// TwinCAT 3 PLC project Untitled3
// ProgramVersion: 3.1.4026.18
// libraries:
//   Tc2_EtherCAT, * (Beckhoff Automation GmbH)
//   Tc2_MC2, * (Beckhoff Automation GmbH)
//   Tc2_Standard, * (Beckhoff Automation GmbH)
//   Tc2_System, * (Beckhoff Automation GmbH)
//   Tc3_EtherCATDiag, * (Beckhoff Automation GmbH)
//   Tc3_EventLogger, * (Beckhoff Automation GmbH)
//   Tc3_Module, * (Beckhoff Automation GmbH)
// project tree:
//   DUTs/ E_SignalMode.TcDUT, ST_TsDiagObjectsEL1904.TcDUT, ST_TsDiagObjectsEL2904.TcDUT, ST_TsDiagObjectsEL1918.TcDUT, ST_TsDiagObjectsEL2912.TcDUT
//   POUs/TwinSAFE FBs/ FB_CoEDiagObjects_EL1904.TcPOU, FB_CoEDiagObjects_EL1918.TcPOU (not stored), FB_CoEDiagObjects_EL2904.TcPOU (not stored), FB_CoEDiagObjects_EL2912.TcPOU (not stored), FB_TsConnection_Diag.TcPOU (not stored), FB_TsConnection_Diag_EL2912.TcPOU, FB_TsConnection_EtherCATState_EL2904.TcPOU, FB_TsConnection_EtherCATState_EL2912.TcPOU, FB_TsConnection_State.TcPOU (not stored), FB_TsConnection_EtherCatState_EL1918.TcPOU, FB_TsConnection_Diag_EL1918.TcPOU, FB_TsConnection_EtherCATState_EL1904.TcPOU (not stored), FB_TsFBEDM_Diag.TcPOU, FB_TsFBEDM_State.TcPOU, FB_TsFBEStop_Diag.TcPOU, FB_TsFBEStop_State.TcPOU (not stored), FB_TsFBMon_Diag.TcPOU (not stored), FB_TsFBMon_State.TcPOU, FB_TsGroup_Diag.TcPOU (not stored), FB_TsGroup_State.TcPOU (not stored)
//   POUs/ MAIN.TcPOU
//   / Test1.TcTTO
// real-time tasks:
//   TASK Test1: cycle T#10ms, priority 2, ADS port 350
// motion (NC):
//   TASK NC-Task 1 SAF NEW: cycle T#2ms, priority 4, ADS port 501
//   TASK NC-Task 1 SVB: cycle T#10ms, priority 8, ADS port 511
//   AXIS Axis 1 (id 1)
//     General: UnitName=°
//     Dynamic: Acceleration=15000, Deceleration=15000, Jerk=52947
//     Velo: RefSearch=117.66, RefSync=117.66, SlowManual=588.3, FastManual=3529.8, Fast=11766, Maximum=11766
//     OtherSettings: AllowMotionCmdToSlave=true
//     encoder EncType=19
//       EncPara: ScaleFactorNumerator=360, ScaleFactorDenominator=1048576, MaxCount=#xffffffff
//     drive DrvType=16
//       DrvPara: MaxCount=#xffffffff, DriveControlDWord=#x00020100
//         Analog: VeloReferenz=12942.6, VeloScale=32, TorqueSetpointScale=10, ScaleFactorActTorque=0.1
//         TimeComp: TaskDelayCycles=1
//     controller CtrType=1
//       CtrPara: PriorControlFactor=1
//         PosDiffControl: Range=50
//         Observer: BandWidth=20
//   AXIS Axis 2 (id 2)
//     General: UnitName=°
//     Dynamic: Acceleration=4263.1575, Deceleration=4263.1575, Jerk=12789.4725
//     Velo: RefSearch=28.42105, RefSync=28.42105, SlowManual=142.10525, FastManual=852.6315, Fast=2842.105, Maximum=2842.105
//     OtherSettings: AllowMotionCmdToSlave=true
//     encoder EncType=4
//       EncPara: ScaleFactorNumerator=360, ScaleFactorDenominator=4096, MaxCount=#x0000ffff
//         Inc: RefSoftSyncMask=#x0000ffff
//     drive DrvType=24
//       Analog: VeloReferenz=3600, TorqueSetpointScale=10, ScaleFactorActTorque=0.1
//       TimeComp: TaskDelayCycles=1
//     controller CtrType=1
//       CtrPara: PriorControlFactor=1
//         PosDiffControl: Range=50
//         Observer: BandWidth=20
// I/O:
//   DEVICE Device 1 (EtherCAT), AmsNetId 169.254.191.109.2.1
//     Term 19 (EK1200) [EK1200-5000 EtherCAT Power supply (2A E-Bus)]
//       Term 20 (EL1918) [EL1918, 8Ch. Safety Input 24V, TwinSAFE]
//         modules: Module 2 (FSLOGIC)
//       Term 21 (EL1904) [EL1904, 4 Ch. Safety Input 24V, TwinSAFE]
//         modules: Module 1 (FSOES)
//       Term 22 (EL2904) [EL2904, 4 Ch. Safety Output 24V, 0.5A, TwinSAFE]
//         modules: Module 1 (FSOES), Module 2 (DO)
//       Term 23 (EK1122) [EK1122 2 port EtherCAT junction]
//         Term 24 (EK1101) [EK1101 EtherCAT Coupler (2A E-Bus, ID switch)]
//           Term 25 (EL2912) [EL2912, 2Ch. Safety Output 24V, 2A, TwinSAFE]
//             modules: Module 1 (FSOE), Module 2 (FSOUT), Module 3 (DEVICEIO), Module 4 (FSLOGIC)
//           Term 26 (EK1122) [EK1122 2 port EtherCAT junction]
//             Term 27 (EK1101-0010) [EK1101-0010 EtherCAT Coupler (2A E-Bus, ID switch, Extended Distance)]
//               Term 28 (EL3074) [EL3074 4Ch. Ana. Input +/-10V, +/-20mA]
//               Term 29 (EL3174) [EL3174 4Ch. Ana. Input +/-10V Diff., +/-20mA SingleEnded, 16 Bit]
//               Term 30 (EL3202-0010) [EL3202-0010 2Ch. Ana. Input PT100 (RTD), High Precision]
//               Term 31 (ELM3142-0000) [ELM3142-0000 2Ch. Ana. Input +/-10V, +/-20mA, 24 bit, high precision]
//               Term 32 (EL4712) [EL4712 2Ch. Ana. Output 0-20mA, Oversample]
//               Term 33 (EL4732) [EL4732 2Ch. Ana. Output +/-10V, Oversample]
//               Term 34 (EL9510) [EL9510 Power supply terminal 10V]
//               Term 35 (EK1122) [EK1122 2 port EtherCAT junction]
//                 Term 36 (EK1100) [EK1100 EtherCAT Coupler (2A E-Bus)]
//                   Term 37 (EL7201-9014) [EL7201-9014 1Ch. MDP742 Servo motor output stage with OCT (50V, 2.8A RMS) and STO input]
//                     startup 32785:21 := 0E01 // DRV Motor Settings / Commutation offset
//                     startup 32785:27 := A9070000 // DRV Motor Settings / Motor speed limitation
//                     startup 28688:3 := 09 // DRV Outputs / Modes of operation
//                     startup 32784:87 := 64 // DRV Amplifier Settings / Velocity feed forward gain
//                     startup 28688:11 := 880B // DRV Outputs / Torque limitation
//                     startup 32784:19 := B200 // DRV Amplifier Settings / Current loop proportional gain
//                     startup 32784:18 := 0500 // DRV Amplifier Settings / Current loop integral time
//                     startup 32784:21 := 2B000000 // DRV Amplifier Settings / Velocity loop proportional gain
//                     startup 32784:20 := 96000000 // DRV Amplifier Settings / Velocity loop integral time
//                     startup 32768:1 := 00 // FB Settings / Invert feedback direction
//                   Term 38 (EL7037) [EL7037 1Ch. Stepper motor output stage (24V, 1.5A)]
//                     startup 32786:5 := 02 // STM Features Ch.1 / Speed range
//                     startup 32785:1 := DE01 // STM Controller Settings Ch.1 / Kp factor (curr.)
//                     startup 32785:2 := A200 // STM Controller Settings Ch.1 / Ki factor (curr.)
//                     startup 32788:3 := C0010000 // STM Controller Settings 3 Ch.1 / Kp factor (velo.)
//                     startup 32788:4 := 8813 // STM Controller Settings 3 Ch.1 / Tn (velo.)
//                     startup 32786:8 := 00 // STM Features Ch.1 / Feedback type
//                   Term 39 (EL9011) [EL9011 End Terminal]
// variable links:
//   Device 1 (EtherCAT) <-> Device 1 (EtherCAT)/Term 19 (EK1200)/Term 21 (EL1904)
//     Term 19 (EK1200)/Term 20 (EL1918)/ConnectionInputs/TwinSafeGroup1.Term 3 (EL1904) - Module 1 (FSOES)_4 TxPDO <-> Module 1 (FSOES)/RxPDO/FSOE
//     Term 19 (EK1200)/Term 20 (EL1918)/ConnectionOutputs/TwinSafeGroup1.Term 3 (EL1904) - Module 1 (FSOES)_4 RxPDO <-> Module 1 (FSOES)/TxPDO/FSOE
//   Device 1 (EtherCAT) <-> Device 1 (EtherCAT)/Term 19 (EK1200)/Term 22 (EL2904)
//     Term 19 (EK1200)/Term 20 (EL1918)/ConnectionInputs/TwinSafeGroup1.Term 4 (EL2904) - Module 1 (FSOES)_5 TxPDO <-> Module 1 (FSOES)/RxPDO/FSOE
//     Term 19 (EK1200)/Term 20 (EL1918)/ConnectionOutputs/TwinSafeGroup1.Term 4 (EL2904) - Module 1 (FSOES)_5 RxPDO <-> Module 1 (FSOES)/TxPDO/FSOE
//   Device 1 (EtherCAT) <-> Device 1 (EtherCAT)/Term 19 (EK1200)/Term 23 (EK1122)/Term 24 (EK1101)/Term 25 (EL2912)
//     Term 19 (EK1200)/Term 20 (EL1918)/ConnectionInputs/TwinSafeGroup1.Term 5 (EL2912) - Module 1 (FSOE)_6 TxPDO <-> Module 1 (FSOE)/FSoE Outputs/FSOE
//     Term 19 (EK1200)/Term 20 (EL1918)/ConnectionOutputs/TwinSafeGroup1.Term 5 (EL2912) - Module 1 (FSOE)_6 RxPDO <-> Module 1 (FSOE)/FSoE Inputs/FSOE
//   NC-Task 1 SAF NEW/Axes/Axis 1 <-> Device 1 (EtherCAT)/Term 19 (EK1200)/Term 23 (EK1122)/Term 24 (EK1101)/Term 26 (EK1122)/Term 27 (EK1101-0010)/Term 35 (EK1122)/Term 36 (EK1100)/Term 37 (EL7201-9014)
//     Drive/Inputs/In/nDataIn1 <-> DRV Following error actual value/Following error actual value
//     Drive/Inputs/In/nDataIn3[0] <-> DRV Torque actual value/Torque actual value
//     Drive/Inputs/In/nDcOutputTime <-> InfoData/DcOutputShift
//     Drive/Inputs/In/nState1 <-> DRV Statusword/Statusword
//     Drive/Inputs/In/nState2 <-> DRV Statusword/Statusword @bit 8
//     Drive/Inputs/In/nState4 @bit 1 <-> WcState/InputToggle
//     Drive/Inputs/In/nState4 <-> WcState/WcState
//     Drive/Outputs/Out/nCtrl1 <-> DRV Controlword/Controlword
//     Drive/Outputs/Out/nCtrl2 <-> DRV Controlword/Controlword @bit 8
//     Drive/Outputs/Out/nDataOut1 <-> DRV Target position/Target position
//     Drive/Outputs/Out/nDataOut2 <-> DRV Target velocity/Target velocity
//     Enc/Inputs/In/nDataIn1 <-> FB Position/Position
//     Enc/Inputs/In/nDcInputTime <-> InfoData/DcInputShift
//     Enc/Inputs/In/nState4 @bit 1 <-> WcState/InputToggle
//     Enc/Inputs/In/nState4 <-> WcState/WcState
//   NC-Task 1 SAF NEW/Axes/Axis 2 <-> Device 1 (EtherCAT)/Term 19 (EK1200)/Term 23 (EK1122)/Term 24 (EK1101)/Term 26 (EK1122)/Term 27 (EK1101-0010)/Term 35 (EK1122)/Term 36 (EK1100)/Term 38 (EL7037)
//     Drive/Inputs/In/nState1 @bit 3 <-> STM Status/Status/Error
//     Drive/Inputs/In/nState1 @bit 7 <-> STM Status/Status/Motor stall
//     Drive/Inputs/In/nState1 @bit 5 <-> STM Status/Status/Moving negative
//     Drive/Inputs/In/nState1 @bit 4 <-> STM Status/Status/Moving positive
//     Drive/Inputs/In/nState1 @bit 1 <-> STM Status/Status/Ready
//     Drive/Inputs/In/nState1 <-> STM Status/Status/Ready to enable
//     Drive/Inputs/In/nState1 @bit 6 <-> STM Status/Status/Torque reduced
//     Drive/Inputs/In/nState1 @bit 2 <-> STM Status/Status/Warning
//     Drive/Inputs/In/nState2 @bit 3 <-> STM Status/Status/Digital input 1
//     Drive/Inputs/In/nState2 @bit 4 <-> STM Status/Status/Digital input 2
//     Drive/Inputs/In/nState2 @bit 5 <-> STM Status/Status/Sync error
//     Drive/Inputs/In/nState2 @bit 7 <-> STM Status/Status/TxPDO Toggle
//     Drive/Inputs/In/nState4 @bit 1 <-> WcState/InputToggle
//     Drive/Inputs/In/nState4 <-> WcState/WcState
//     Drive/Outputs/Out/nCtrl1 <-> STM Control/Control/Enable
//     Drive/Outputs/Out/nCtrl1 @bit 2 <-> STM Control/Control/Reduce torque
//     Drive/Outputs/Out/nCtrl1 @bit 1 <-> STM Control/Control/Reset
//     Drive/Outputs/Out/nCtrl2 @bit 3 <-> STM Control/Control/Digital output 1
//     Drive/Outputs/Out/nDataOut2[0] <-> STM Velocity/Velocity
//     Enc/Inputs/In/nDataIn1[0] <-> ENC Status compact/Counter value
//     Enc/Inputs/In/nDataIn2[0] <-> ENC Status compact/Latch value
//     Enc/Inputs/In/nState1 @bit 4 <-> ENC Status compact/Status/Counter overflow
//     Enc/Inputs/In/nState1 @bit 3 <-> ENC Status compact/Status/Counter underflow
//     Enc/Inputs/In/nState1 @bit 7 <-> ENC Status compact/Status/Extrapolation stall
//     Enc/Inputs/In/nState1 <-> ENC Status compact/Status/Latch C valid
//     Enc/Inputs/In/nState1 @bit 1 <-> ENC Status compact/Status/Latch extern valid
//     Enc/Inputs/In/nState1 @bit 2 <-> ENC Status compact/Status/Set counter done
//     Enc/Inputs/In/nState2 @bit 4 <-> ENC Status compact/Status/Status of extern latch
//     Enc/Inputs/In/nState2 <-> ENC Status compact/Status/Status of input A
//     Enc/Inputs/In/nState2 @bit 1 <-> ENC Status compact/Status/Status of input B
//     Enc/Inputs/In/nState2 @bit 2 <-> ENC Status compact/Status/Status of input C
//     Enc/Inputs/In/nState2 @bit 5 <-> ENC Status compact/Status/Sync error
//     Enc/Inputs/In/nState2 @bit 7 <-> ENC Status compact/Status/TxPDO Toggle
//     Enc/Inputs/In/nState4 @bit 1 <-> WcState/InputToggle
//     Enc/Inputs/In/nState4 <-> WcState/WcState
//     Enc/Outputs/Out/nCtrl1 <-> ENC Control compact/Control/Enable latch C
//     Enc/Outputs/Out/nCtrl1 @bit 3 <-> ENC Control compact/Control/Enable latch extern on negative edge
//     Enc/Outputs/Out/nCtrl1 @bit 1 <-> ENC Control compact/Control/Enable latch extern on positive edge
//     Enc/Outputs/Out/nCtrl1 @bit 2 <-> ENC Control compact/Control/Set counter
//     Enc/Outputs/Out/nDataOut1[0] <-> ENC Control compact/Set counter value
//   Untitled3/Untitled3 Instance <-> Device 1 (EtherCAT)/Term 19 (EK1200)/Term 20 (EL1918)
//     Test1 Inputs/MAIN.bSafety_ComErr <-> StandardInputs/Standard Out Var 8
//     Test1 Inputs/MAIN.bSafety_FBErr <-> StandardInputs/Standard Out Var 7
//     Test1 Inputs/MAIN.bTsModulError1 <-> Device Info Data/Internal I/O/Input Safe Data FSIN Module 1.Module Fault
//     Test1 Inputs/MAIN.bWcState_EL1918 <-> WcState/WcState
//     Test1 Inputs/MAIN.nDiag_EL1904 <-> Connection Info Data/TwinSafeGroup1.Term 3 (EL1904) - Module 1 (FSOES)_4 Info Data/Diag
//     Test1 Inputs/MAIN.nDiag_EL2904 <-> Connection Info Data/TwinSafeGroup1.Term 4 (EL2904) - Module 1 (FSOES)_5 Info Data/Diag
//     Test1 Inputs/MAIN.nDiag_EL2912 <-> Connection Info Data/TwinSafeGroup1.Term 5 (EL2912) - Module 1 (FSOE)_6 Info Data/Diag
//     Test1 Inputs/MAIN.nDiag_TsFBEDM <-> Function Block Info Data/TwinSafeGroup1.Network1_EStop.FBEdm1 Info Data/Diag
//     Test1 Inputs/MAIN.nDiag_TsFBEstop <-> Function Block Info Data/TwinSafeGroup1.Network1_EStop.FBEstop1 Info Data/Diag
//     Test1 Inputs/MAIN.nDiag_TsFBMon <-> Function Block Info Data/TwinSafeGroup1.Network2_MON.FBMon1 Info Data/Diag
//     Test1 Inputs/MAIN.nDiag_TsGroup1 <-> TwinSAFE Group Info Data/TwinSafeGroup1 Info Data/Diag
//     Test1 Inputs/MAIN.nEtherCATState_EL1918 <-> InfoData/State
//     Test1 Inputs/MAIN.nState_EL1904 <-> Connection Info Data/TwinSafeGroup1.Term 3 (EL1904) - Module 1 (FSOES)_4 Info Data/State
//     Test1 Inputs/MAIN.nState_EL2904 <-> Connection Info Data/TwinSafeGroup1.Term 4 (EL2904) - Module 1 (FSOES)_5 Info Data/State
//     Test1 Inputs/MAIN.nState_EL2912 <-> Connection Info Data/TwinSafeGroup1.Term 5 (EL2912) - Module 1 (FSOE)_6 Info Data/State
//     Test1 Inputs/MAIN.nState_TsFBEDM <-> Function Block Info Data/TwinSafeGroup1.Network1_EStop.FBEdm1 Info Data/State
//     Test1 Inputs/MAIN.nState_TsFBEstop <-> Function Block Info Data/TwinSafeGroup1.Network1_EStop.FBEstop1 Info Data/State
//     Test1 Inputs/MAIN.nState_TsFBMon <-> Function Block Info Data/TwinSafeGroup1.Network2_MON.FBMon1 Info Data/State
//     Test1 Inputs/MAIN.nState_TsGroup1 <-> TwinSAFE Group Info Data/TwinSafeGroup1 Info Data/State
//     Test1 Outputs/MAIN.bSafery_RestartEStop <-> StandardOutputs/Standard In Var 10
//     Test1 Outputs/MAIN.bSafery_RestartMON <-> StandardOutputs/Standard In Var 12
//     Test1 Outputs/MAIN.bSafety_ErrAck <-> StandardOutputs/Standard In Var 1
//     Test1 Outputs/MAIN.bSafety_RunStop <-> StandardOutputs/Standard In Var 2
//   Untitled3/Untitled3 Instance <-> Device 1 (EtherCAT)/Term 19 (EK1200)/Term 21 (EL1904)
//     Test1 Inputs/MAIN.bWcState_EL1904 <-> WcState/WcState
//     Test1 Inputs/MAIN.nEtherCATState_EL1904 <-> InfoData/State
//   Untitled3/Untitled3 Instance <-> Device 1 (EtherCAT)/Term 19 (EK1200)/Term 22 (EL2904)
//     Test1 Inputs/MAIN.bWcState_EL2904 <-> WcState/WcState
//     Test1 Inputs/MAIN.nEtherCATState_EL2904 <-> InfoData/State
//   Untitled3/Untitled3 Instance <-> Device 1 (EtherCAT)/Term 19 (EK1200)/Term 23 (EK1122)/Term 24 (EK1101)/Term 25 (EL2912)
//     Test1 Inputs/MAIN.bWcState_EL2912_1 <-> WcState/WcState0
//     Test1 Inputs/MAIN.bWcState_EL2912_2 <-> WcState/WcState1
//     Test1 Inputs/MAIN.nEtherCATState_EL2912 <-> InfoData/State
//   Untitled3/Untitled3 Instance <-> Device 1 (EtherCAT)/Term 19 (EK1200)/Term 23 (EK1122)/Term 24 (EK1101)/Term 26 (EK1122)/Term 27 (EK1101-0010)/Term 28 (EL3074)
//     Test1 Inputs/MAIN.EL3074.MDP5001_300_Input/MDP5001_300_AI_Standard_Channel_1_Status/Error <-> AI Standard Channel 1/Status/Error
//     Test1 Inputs/MAIN.EL3074.MDP5001_300_Input/MDP5001_300_AI_Standard_Channel_1_Status/Overrange <-> AI Standard Channel 1/Status/Overrange
//     Test1 Inputs/MAIN.EL3074.MDP5001_300_Input/MDP5001_300_AI_Standard_Channel_1_Status/Underrange <-> AI Standard Channel 1/Status/Underrange
//     Test1 Inputs/MAIN.nIn3074V1 <-> AI Standard Channel 1/Value
//   Untitled3/Untitled3 Instance <-> Device 1 (EtherCAT)/Term 19 (EK1200)/Term 23 (EK1122)/Term 24 (EK1101)/Term 26 (EK1122)/Term 27 (EK1101-0010)/Term 29 (EL3174)
//     Test1 Inputs/MAIN.EL3174.MDP5001_300_Input/MDP5001_300_AI_Standard_Channel_1_Status/Error <-> AI Standard Channel 1/Status/Error
//     Test1 Inputs/MAIN.EL3174.MDP5001_300_Input/MDP5001_300_AI_Standard_Channel_1_Status/Overrange <-> AI Standard Channel 1/Status/Overrange
//     Test1 Inputs/MAIN.EL3174.MDP5001_300_Input/MDP5001_300_AI_Standard_Channel_1_Status/Underrange <-> AI Standard Channel 1/Status/Underrange
//     Test1 Inputs/MAIN.nIn3174A1 <-> AI Standard Channel 1/Value
//   Untitled3/Untitled3 Instance <-> Device 1 (EtherCAT)/Term 19 (EK1200)/Term 23 (EK1122)/Term 24 (EK1101)/Term 26 (EK1122)/Term 27 (EK1101-0010)/Term 30 (EL3202-0010)
//     Test1 Inputs/MAIN.EL3202.MDP5001_320_Input/MDP5001_320_RTD_Inputs_Channel_1_Status/Error <-> RTD Inputs Channel 1/Status/Error
//     Test1 Inputs/MAIN.EL3202.MDP5001_320_Input/MDP5001_320_RTD_Inputs_Channel_1_Status/Overrange <-> RTD Inputs Channel 1/Status/Overrange
//     Test1 Inputs/MAIN.EL3202.MDP5001_320_Input/MDP5001_320_RTD_Inputs_Channel_1_Status/Underrange <-> RTD Inputs Channel 1/Status/Underrange
//     Test1 Inputs/MAIN.nRTD <-> RTD Inputs Channel 1/Value
//   Untitled3/Untitled3 Instance <-> Device 1 (EtherCAT)/Term 19 (EK1200)/Term 23 (EK1122)/Term 24 (EK1101)/Term 26 (EK1122)/Term 27 (EK1101-0010)/Term 31 (ELM3142-0000)
//     Test1 Inputs/MAIN.ELM3142.MDP5001_350_Input/MDP5001_350_PAI_Status_Channel_1_Status/Error <-> PAI Status Channel 1/Status/Error
//     Test1 Inputs/MAIN.ELM3142.MDP5001_350_Input/MDP5001_350_PAI_Status_Channel_1_Status/Overrange <-> PAI Status Channel 1/Status/Overrange
//     Test1 Inputs/MAIN.ELM3142.MDP5001_350_Input/MDP5001_350_PAI_Status_Channel_1_Status/Underrange <-> PAI Status Channel 1/Status/Underrange
//     Test1 Inputs/MAIN.nELM <-> PAI Samples 1 Channel 1/Samples[0]
//   Untitled3/Untitled3 Instance <-> Device 1 (EtherCAT)/Term 19 (EK1200)/Term 23 (EK1122)/Term 24 (EK1101)/Term 26 (EK1122)/Term 27 (EK1101-0010)/Term 32 (EL4712)
//     Test1 Outputs/MAIN.nOutA1 <-> Ch1 Sample 0/Ch1 Value
//   Untitled3/Untitled3 Instance <-> Device 1 (EtherCAT)/Term 19 (EK1200)/Term 23 (EK1122)/Term 24 (EK1101)/Term 26 (EK1122)/Term 27 (EK1101-0010)/Term 33 (EL4732)
//     Test1 Outputs/MAIN.nOutV1 <-> Ch1 Sample 0/Ch1 Value
//   Untitled3/Untitled3 Instance <-> NC-Task 1 SAF NEW/Axes/Axis 1
//     Test1 Inputs/MAIN.Axis1.NcToPlc <-> Outputs/ToPlc
//     Test1 Outputs/MAIN.Axis1.PlcToNc <-> Inputs/FromPlc
//   Untitled3/Untitled3 Instance <-> NC-Task 1 SAF NEW/Axes/Axis 2
//     Test1 Inputs/MAIN.Axis2.NcToPlc <-> Outputs/ToPlc
//     Test1 Outputs/MAIN.Axis2.PlcToNc <-> Inputs/FromPlc

CONFIGURATION Untitled3
    RESOURCE PLC ON TwinCAT3
        TASK Test1(INTERVAL := T#10ms, PRIORITY := 2);
        PROGRAM MAIN WITH Test1 : MAIN;
    END_RESOURCE
END_CONFIGURATION

// ---- DUTs/E_SignalMode.TcDUT
TYPE E_SignalMode :
(

	SignalMode_Off,
    SignalMode_Static,
    SignalMode_Rectangle,
    SignalMode_Sinus,
    SignalMode_Triangle
   
);
END_TYPE

// ---- DUTs/ST_TsDiagObjectsEL1904.TcDUT
TYPE ST_TsDiagObjectsEL1904 :
(*******************************************************************************************************
Description			:	Index 16#800E Diagnostic objects
Supported terminals : 	EL1904
********************************************************************************************************)
STRUCT

	nNotUsedData1								:ARRAY[0..8] OF UINT;

(* Sensor test error *)
	nSensorTestError						:UINT;
	(*TsDiagObjectsBitsEL1904_bSensorTestError_Input1		 		:= stDiagObjects.nSensorTestError.0;
	TsDiagObjectsBitsEL1904_bSensorTestError_Input2		 			 := stDiagObjects.nSensorTestError.1;
	TsDiagObjectsBitsEL1904_bSensorTestError_Input3		 			 := stDiagObjects.nSensorTestError.2;
	TsDiagObjectsBitsEL1904_bSensorTestError_Input4		 			 := stDiagObjects.nSensorTestError.3;*)
	

(* Error during two channel evaluation *)
	nDuringTwoChannelEvaluationError		:UINT;
	(*TsDiagObjectsBitsEL1904_bErrFirstInputPair 			 := stDiagObjects.nDuringTwoChannelEvaluationError.0;
	TsDiagObjectsBitsEL1904_bErrSecondInputPair 		 := stDiagObjects.nDuringTwoChannelEvaluationError.1;*)


(* Error in the safety mat operating mode: input pair disagree *)
	nMatModeInputPairDisagreeError			:UINT;
	(*TsDiagObjectsBitsEL1904_bMatOpModeErrFirstInputPair	 := stDiagObjects.nMatModeInputPairDisagreeError.0 
																			AND stDiagObjects.nMatModeInputPairDisagreeError.1;
	TsDiagObjectsBitsEL1904_bMatOpModeErrSecondInputPair := stDiagObjects.nMatModeInputPairDisagreeError.2 
																			AND stDiagObjects.nMatModeInputPairDisagreeError.3;*)
	
(* Error in the safety mat operating mode: external supply *)
	nMatModeExternalSupplyError				:UINT;
	(*TsDiagObjectsBitsEL1904_bMatOpModeExtSupplyError_Input1 := stDiagObjects.nMatModeExternalSupplyError.0;
	TsDiagObjectsBitsEL1904_bMatOpModeExtSupplyError_Input2 := stDiagObjects.nMatModeExternalSupplyError.1;
	TsDiagObjectsBitsEL1904_bMatOpModeExtSupplyError_Input3 := stDiagObjects.nMatModeExternalSupplyError.2;
	TsDiagObjectsBitsEL1904_bMatOpModeExtSupplyError_Input4 := stDiagObjects.nMatModeExternalSupplyError.3;*)
	
	nNotUsedData2								:ARRAY[0..2] OF UINT;

END_STRUCT
END_TYPE
(* End *)

// ---- DUTs/ST_TsDiagObjectsEL2904.TcDUT
TYPE ST_TsDiagObjectsEL2904 :
(*******************************************************************************************************
Description			:	Index 16#800E Diagnostic objects
Supported terminals : 	EL1904
********************************************************************************************************)
STRUCT

	nNotUsedData1								:ARRAY[0..8] OF UINT;

(* Sensor test error *)
	nSensorTestError						:UINT;
	(*TsDiagObjectsBitsEL2904_bSensorTestError_Output1		 		  	 := stDiagObjects.nSensorTestError.0;
	TsDiagObjectsBitsEL2904_bSensorTestError_Output2		 			 := stDiagObjects.nSensorTestError.1;
	TsDiagObjectsBitsEL2904_bSensorTestError_Output3		 			 := stDiagObjects.nSensorTestError.2;
	TsDiagObjectsBitsEL2904_bSensorTestError_Output4		 			 := stDiagObjects.nSensorTestError.3;*)
	


(* Error in the safety mat operating mode: input pair disagree *)
	nMatModeInputPairDisagreeError			:UINT;
	(*TsDiagObjectsBitsEL2904_bMatOpModeErrFirstInputPair	 := stDiagObjects.nMatModeInputPairDisagreeError.0 
																			AND stDiagObjects.nMatModeInputPairDisagreeError.1;
	TsDiagObjectsBitsEL2904_bMatOpModeErrSecondInputPair := stDiagObjects.nMatModeInputPairDisagreeError.2 
																			AND stDiagObjects.nMatModeInputPairDisagreeError.3;*)
	
(* Error in the safety mat operating mode: external supply *)
	nMatModeExternalSupplyError				:UINT;
	(*TsDiagObjectsBitsEL2904_bMatOpModeExtSupplyError_Output1 := stDiagObjects.nMatModeExternalSupplyError.0;
	TsDiagObjectsBitsEL2904_bMatOpModeExtSupplyError_Output2 := stDiagObjects.nMatModeExternalSupplyError.1;
	TsDiagObjectsBitsEL2904_bMatOpModeExtSupplyError_Output3 := stDiagObjects.nMatModeExternalSupplyError.2;
	TsDiagObjectsBitsEL2904_bMatOpModeExtSupplyError_Output4 := stDiagObjects.nMatModeExternalSupplyError.3;*)
	
	nNotUsedData2								:ARRAY[0..2] OF UINT;

END_STRUCT
END_TYPE
(* End *)

// ---- DUTs/ST_TsDiagObjectsEL1918.TcDUT
TYPE ST_TsDiagObjectsEL1918 :
(*******************************************************************************************************
Description			:	Index 16#800E Diagnostic objects
Supported terminals : 	EL1918
********************************************************************************************************)
STRUCT

	nNotUsedData1								:ARRAY[0..8] OF UINT;

(* Sensor test error *)
	nSensorTestError						:UINT;
	(*TsDiagObjectsBitsEL1918_bSensorTestError_Input1		 		:= stDiagObjects.nSensorTestError.0;
	TsDiagObjectsBitsEL1918_bSensorTestError_Input2		 			 := stDiagObjects.nSensorTestError.1;
	TsDiagObjectsBitsEL1918_bSensorTestError_Input3		 			 := stDiagObjects.nSensorTestError.2;
	TsDiagObjectsBitsEL1918_bSensorTestError_Input4		 			 := stDiagObjects.nSensorTestError.3;*)
	

(* Error during two channel evaluation *)
	nDuringTwoChannelEvaluationError		:UINT;
	(*TsDiagObjectsBitsEL1918_bErrFirstInputPair 			 := stDiagObjects.nDuringTwoChannelEvaluationError.0;
	TsDiagObjectsBitsEL1918_bErrSecondInputPair 		 := stDiagObjects.nDuringTwoChannelEvaluationError.1;*)


(* Error in the safety mat operating mode: input pair disagree *)
	nMatModeInputPairDisagreeError			:UINT;
	(*TsDiagObjectsBitsEL1918_bMatOpModeErrFirstInputPair	 := stDiagObjects.nMatModeInputPairDisagreeError.0 
																			AND stDiagObjects.nMatModeInputPairDisagreeError.1;
	TsDiagObjectsBitsEL1918_bMatOpModeErrSecondInputPair := stDiagObjects.nMatModeInputPairDisagreeError.2 
																			AND stDiagObjects.nMatModeInputPairDisagreeError.3;*)
	
(* Error in the safety mat operating mode: external supply *)
	nMatModeExternalSupplyError				:UINT;
	(*TsDiagObjectsBitsEL1918_bMatOpModeExtSupplyError_Input1 := stDiagObjects.nMatModeExternalSupplyError.0;
	TsDiagObjectsBitsEL1918_bMatOpModeExtSupplyError_Input2 := stDiagObjects.nMatModeExternalSupplyError.1;
	TsDiagObjectsBitsEL1918_bMatOpModeExtSupplyError_Input3 := stDiagObjects.nMatModeExternalSupplyError.2;
	TsDiagObjectsBitsEL1918_bMatOpModeExtSupplyError_Input4 := stDiagObjects.nMatModeExternalSupplyError.3;*)
	
	nNotUsedData2								:ARRAY[0..2] OF UINT;

END_STRUCT
END_TYPE
(* End *)

// ---- DUTs/ST_TsDiagObjectsEL2912.TcDUT
TYPE ST_TsDiagObjectsEL2912 :
(*******************************************************************************************************
Description			:	Index 16#800E Diagnostic objects
Supported terminals : 	EL1904
********************************************************************************************************)
STRUCT

	nNotUsedData1								:ARRAY[0..8] OF UINT;

(* Sensor test error *)
	nSensorTestError						:UINT;
	(*TsDiagObjectsBitsEL2904_bSensorTestError_Output1		 		  	 := stDiagObjects.nSensorTestError.0;
	TsDiagObjectsBitsEL2904_bSensorTestError_Output2		 			 := stDiagObjects.nSensorTestError.1;
	TsDiagObjectsBitsEL2904_bSensorTestError_Output3		 			 := stDiagObjects.nSensorTestError.2;
	TsDiagObjectsBitsEL2904_bSensorTestError_Output4		 			 := stDiagObjects.nSensorTestError.3;*)
	


(* Error in the safety mat operating mode: input pair disagree *)
	nMatModeInputPairDisagreeError			:UINT;
	(*TsDiagObjectsBitsEL2904_bMatOpModeErrFirstInputPair	 := stDiagObjects.nMatModeInputPairDisagreeError.0 
																			AND stDiagObjects.nMatModeInputPairDisagreeError.1;
	TsDiagObjectsBitsEL2904_bMatOpModeErrSecondInputPair := stDiagObjects.nMatModeInputPairDisagreeError.2 
																			AND stDiagObjects.nMatModeInputPairDisagreeError.3;*)
	
(* Error in the safety mat operating mode: external supply *)
	nMatModeExternalSupplyError				:UINT;
	(*TsDiagObjectsBitsEL2904_bMatOpModeExtSupplyError_Output1 := stDiagObjects.nMatModeExternalSupplyError.0;
	TsDiagObjectsBitsEL2904_bMatOpModeExtSupplyError_Output2 := stDiagObjects.nMatModeExternalSupplyError.1;
	TsDiagObjectsBitsEL2904_bMatOpModeExtSupplyError_Output3 := stDiagObjects.nMatModeExternalSupplyError.2;
	TsDiagObjectsBitsEL2904_bMatOpModeExtSupplyError_Output4 := stDiagObjects.nMatModeExternalSupplyError.3;*)
	
	nNotUsedData2								:ARRAY[0..2] OF UINT;

END_STRUCT
END_TYPE
(* End *)

// ---- POUs/MAIN.TcPOU
PROGRAM MAIN
VAR
	
//////////////////////////////////////////////////////TWINSAFE/////////////////////////////////////////////////////////////////////////////////

//Fabian

	//Variables for running the safety project
	bSafety_RunStop					AT%Q*	: BOOL;
	bSafety_ErrAck					AT%Q*	: BOOL;
	bSafery_RestartEStop			AT%Q*	: BOOL;
	bSafery_RestartMON				AT%Q*	: BOOL;
	bSafety_FBErr					AT%I*	: BOOL;
	bSafety_ComErr					AT%I*	: BOOL;
	

	
	//Variables for the error analysis
	fbEcCoeSdoRead							: FB_EcCoESdoReadEx;
	fbTsConnectionState						: FB_TsConnection_State;
	fbTsConnectionDiag						: FB_TsConnection_Diag;
	stDiagObjects							: ST_TsDiagObjectsEL1904;
	fbCoEDiagObjectsEL1904					: FB_CoEDiagObjects_EL1904;
	sErrorText_EL1904						: STRING(255);
	stDiagObjectsEL1918						: ST_TsDiagObjectsEL1918;
	fbCoEDiagObjectsEL1918					: FB_CoEDiagObjects_EL1918;
	sErrorText_EL1918						: STRING(255);
	stDiagObjectsEL2904						: ST_TsDiagObjectsEL2904;
	fbCoEDiagObjectsEL2904					: FB_CoEDiagObjects_EL2904;
	sErrorText_EL2904						: STRING(255);
	stDiagObjectsEL2912						: ST_TsDiagObjectsEL2912;
	fbCoEDiagObjectsEL2912					: FB_CoEDiagObjects_EL2912;
	sErrorText_EL2912						: STRING(255);
	
	//Specific TwinSAFE Module related variables
	bTsModulError1					AT%I*	: BOOL;
	sDiagModulError1						: STRING;
	
	//Specific TwinSAFE group related variables
	fbTsGroupState							: FB_TsGroup_State;
	fbTsGroupDiag							: FB_TsGroup_Diag;
	nState_TsGroup1					AT%I*	: USINT;
	sState_TsGroup1							: STRING(255);
	nDiag_TsGroup1					AT%I*	: USINT;
	sDiag_TsGroup1							: STRING;
	
	//Specific TwinSAFE FBs related variables
	fbTsFBEdmState							: FB_TsFBEDM_State;
	fbTsFBEdmDiag							: FB_TsFBEDM_Diag;
	nState_TsFBEDM					AT%I*	: USINT;
	sState_TsFBEDM							: STRING(255);
	nDiag_TsFBEDM					AT%I*	: USINT;
	sDiag_TsFBEDM							: STRING(255);
	fbTsFBEstopState						: FB_TsFBEStop_State;
	fbTsFBEstopDiag							: FB_TsFBEStop_Diag;
	nState_TsFBEstop				AT%I*	: USINT;
	sState_TsFBEstop						: STRING(255);
	nDiag_TsFBEstop					AT%I*	: UINT;
	sDiag_TsFBEstop							: STRING(255);
	fbTsFBMonState							: FB_TsFBMon_State;
	fbTsFBMonDiag							: FB_TsFBMon_Diag;
	nState_TsFBMon					AT%I*	: USINT;
	sState_TsFBMon							: STRING(255);
	nDiag_TsFBMon					AT%I*	: UINT;
	sDiag_TsFBMon							: STRING(255);
	
	//Specific TwinSAFE terminal related variables
		// EL1904
	fbTsConnectionStateEL1904 				: FB_TsConnection_EtherCatState_EL1904;
 // fbTsConnectionDiagEL1904  				: FB_TsConnection_Diag_EL1904;
	nEtherCATState_EL1904			AT%I*	: UINT;
	sEtherCATState_EL1904					: STRING(255);
	bWcState_EL1904					AT%I*	: BOOL;
	nState_EL1904					AT%I*	: USINT;
	sState_EL1904							: STRING(255);
	nDiag_EL1904					AT%I*	: USINT;
	sDiagPart1_EL1904						: STRING(255);
	sDiagPart2_EL1904						: STRING(255);
		// EL1918
	nEtherCATState_EL1918			AT%I*	: UINT;
	sEtherCATState_EL1918					: STRING(255);
	bWcState_EL1918					AT%I*	: BOOL;
	nState_EL1918					AT%I*	: USINT;
	sState_EL1918							: STRING(255);
	nDiag_EL1918					AT%I*	: USINT;
	sDiagPart1_EL1918						: STRING(255);
	sDiagPart2_EL1918						: STRING(255);
	fbTsConnectionStateEL1918 				: FB_TsConnection_EtherCatState_EL1918;
    fbTsConnectionDiagEL1918  				: FB_TsConnection_Diag_EL1918;
	sStateTextEL1918 						: STRING(50);
    sDiagTextEL1918  						: STRING(255);
    sFullTextEL1918  						: STRING(300);
		// EL2904
	nEtherCATState_EL2904			AT%I*	: UINT;
	sEtherCATState_EL2904					: STRING(255);
	fbTsConnectionStateEL2904 				: FB_TsConnection_EtherCatState_EL2904;
   // fbTsConnectionDiagEL2904  				: FB_TsConnection_Diag_EL2904;
	bWcState_EL2904					AT%I*	: BOOL;
	nState_EL2904					AT%I*	: USINT;
	sState_EL2904							: STRING(255);
	nDiag_EL2904					AT%I*	: USINT;
	sDiagPart1_EL2904						: STRING(255);
	sDiagPart2_EL2904						: STRING(255);
		// EL2912
	nEtherCATState_EL2912			AT%I*	: UINT;
	sEtherCATState_EL2912					: STRING(255);
	fbTsConnectionStateEL2912				: FB_TsConnection_EtherCatState_EL2912;
 	fbTsConnectionDiagEL2912  				: FB_TsConnection_Diag_EL2912;
	sStateTextEL2912 						: STRING(50);
	sDiagTextEL2912  						: STRING(255);
	bWcState_EL2912_1				AT%I*	: BOOL;
	bWcState_EL2912_2				AT%I*	: BOOL;
	nState_EL2912					AT%I*	: USINT;
	sState_EL2912							: STRING(255);
	nDiag_EL2912					AT%I*	: USINT;
	sDiagPart1_EL2912						: STRING(255);
	sDiagPart2_EL2912						: STRING(255);
	
	//Additional variables
	MasterAmsNetID				AT%I*		: T_AmsNetIdArr;
	sMasterNetID							: T_AmsNetId;
	
	
	sErrorTextPopup							: STRING(255);
	sErrorTextPopup2						: STRING(255);
	sErrorTextPopup3						: STRING(255);
	bInitDone 								: BOOL			:= FALSE;
	nCount									: REAL;
	nCount2									: REAL;
	
//////////////////////////////////////////////////////Analog/////////////////////////////////////////////////////////////////////////////////

//Dogan

    bExecute        : BOOL;
	nElmCurr			: REAL;
	
	// Fehlerbits
	EL3074				: MDP5001_300_E23EC103;
	EL3074_Underrange	: BOOL;
	EL3074_Overrange	: BOOL;
	EL3074_Error		: BOOL;
	
	EL3174 				: MDP5001_300_B3F675AA;
	AI3174_Underrange 	: BOOL;
    AI3174_Overrange  	: BOOL;
    AI3174_Error      	: BOOL;
	
	ELM3142				: MDP5001_350_03DC4FA7;
	ELM3142_Underrange 	: BOOL;
    ELM3142_Overrange  	: BOOL;
    ELM3142_Error      	: BOOL;
	
	EL3202				: MDP5001_320_65048876;
	EL3202_Underrange	: BOOL;
	EL3202_Overrange	: BOOL;
	EL3202_Error		: BOOL;
    // Ein-/Ausgänge
    nOutV1          AT%Q* : INT;
    nIn3074V1       AT%I* : INT;
	nOutA1			AT%Q* : INT;
	nIn3174A1		AT%I* : INT;
	nRTD			AT%I* : INT;
	nELM			AT%I* : DINT;
	nRTDVal					: REAL;
	nCurr					: REAL;
	nVoltELM				: LREAL;
	nVoltEL					: REAL;
    // Umschaltung der Signalart
    SignalMode      : E_SignalMode := SignalMode_Off;
    // Rechtecksignal
    tOn             : TON;
    bOut            : BOOL;
    // Sinussignal
    fAmplitude      : REAL := 30000.0; 
    fFrequency      : REAL := 1.0;  
    fOffset         : REAL := 0.0;     
    fSinusValue     : REAL;
    tNow            : TIME;
    tLastCycle      : TIME;
    fTime           : REAL := 0.0;
	bLastExecute    : BOOL := FALSE; // Merker für Flankenwechsel
	
	//Dreiecksignal
    fPeriod     : REAL := 1.0;              // Dauer einer Periode in Sekunden
    fSlope      : REAL;
    fPhase      : REAL;
    fTriangle   : REAL;

//Alarm
	fbEventlogger : FB_TcEventLogger;
	fbAlarm: FB_TcAlarm;
	fbMessage: FB_TcMessage;
	
	bAlarm: BOOL;
	bMessage : BOOL;
	bIsInitalized: BOOL;
	bClearAlarm: BOOL;
	bConfirmAlarm: BOOL;
	
	bClearLoggedEvents: BOOL;
	ClearLoggedEvents: INT;
	
	

//////////////////////////////////////////////////////Motion/////////////////////////////////////////////////////////////////////////////////

//Kuba
	
	//AXIS1 -Servomotor-
	Axis1 : AXIS_ref;
	fbPower	: MC_Power;
	bEnable		: BOOL;
	fbReset	: MC_Reset;
	bReset		: BOOL;
	fbMoveVelocity	: MC_MoveVelocity;
	bMove		: BOOL;
	
	//Fehlermeldung
	fbReadDiag : FB_CoE_DiagHistory_ReadAxis;
	bRead : BOOL;
	aMessages : ARRAY [0..10] OF ST_CoE_DiagHistory_Entry;
	nCase: INT;
	bStartSequence: BOOL;
	
	//AXIS2 -Steppermotor-
	Axis2 : AXIS_REF;
	fbPower2 : MC_Power;
	fbReset2 : MC_Reset;
	fbMoveVelocity2	: MC_MoveVelocity;
	
	bEnable2 : BOOL;
	bReset2 : BOOL;
	bMove2 : BOOL;
	
	//Fehlermeldung
	fbReadDiag2 : FB_CoE_DiagHistory_ReadAxis;
	bRead2 : BOOL;
	aMessages2 : ARRAY [0..10] OF ST_CoE_DiagHistory_Entry;
	nCase2: INT;
	bStartSequence2: BOOL;
	
	//ALLGEMEINE
	nVelocity: LREAL := 360;
	nDynamik: LREAL := 1000;
	nDynamik2: LREAL := 1000;
	
	
END_VAR



//////////////////////////////////////////////////////TWINSAFE/////////////////////////////////////////////////////////////////////////////////

//Fabian
(*
bSafety_RunStop := TRUE;

nCount := nCount +0.1;
IF nCount >= 170 THEN
	nCount := 0;
END_IF

nCount2 := nCount2 -0.0765;
IF nCount2 <= -130 THEN
	nCount2 := 0;
END_IF

sDiagPart1_EL1918 := 'No Error detacted';
sDiagPart2_EL1918 := '';
sErrorText_EL1918 := '';

// EL1904
sDiagPart1_EL1904 := 'No Error detacted';
sDiagPart2_EL1904 := '';
sErrorText_EL1904 := '';

// EL2904
sDiagPart1_EL2904 := 'No Error detacted';
sDiagPart2_EL2904 := '';
sErrorText_EL2904 := '';

// EL2912
sDiagPart1_EL2912 := 'No Error detacted';
sDiagPart2_EL2912 := '';
sErrorText_EL2912 := '';

//bInitDone := TRUE; // nur einmal ausführen

//group state of TwinSAFE Group 1
fbTsGroupState(nState:=nState_TsGroup1);
sState_TsGroup1 := fbTsGroupState.sState; 	//writing the actual group state as text into a string variable

//Device EtherCAT State
	//EL1918
		fbTsConnectionStateEL1918(nEtherCATState := nEtherCATState_EL1918);
		sEtherCATState_EL1918 := fbTsConnectionStateEL1918.sEtherCATState;
	//EL1904
		fbTsConnectionStateEL1904(nEtherCATState := nEtherCATState_EL1904);
		sEtherCATState_EL1904 := fbTsConnectionStateEL1904.sEtherCATState;	
	//EL2904
		fbTsConnectionStateEL2904(nEtherCATState := nEtherCATState_EL2904);
		sEtherCATState_EL2904 := fbTsConnectionStateEL2904.sEtherCATState;		
	//EL2912
		fbTsConnectionStateEL2912(nEtherCATState := nEtherCATState_EL2912);
		sEtherCATState_EL2912 := fbTsConnectionStateEL2912.sEtherCATState;		
//Device FSoE State
	//EL1918
	
	//EL1904
		fbTsConnectionStateEL1918(nEtherCATState := nEtherCATState_EL1918);
		sEtherCATState_EL1918 := fbTsConnectionStateEL1918.sEtherCATState;
		fbTsConnectionState(nState:=nState_EL1904);
		sState_EL1904 := fbTsConnectionState.sState;
	//EL2904
		fbTsConnectionState(nState:=nState_EL2904);
		sState_EL2904 := fbTsConnectionState.sState;
	//EL2912
		fbTsConnectionState(nState:=nState_EL2912);
		sState_EL2912 := fbTsConnectionState.sState;
//group diag of TwinSAFE Group 1
fbTsGroupDiag(nDiag:=nDiag_TsGroup1);
sDiag_TsGroup1 := fbTsGroupDiag.sDiag;		//writing the actual group diag as text into a string variable


IF bTsModulError1 THEN
		sDiagModulError1 := 'EL1918 0x8062 SAFEIN:Diagnosis Test: Feedback in Step2 active Channel is wrong. Module:0x3 / DiagChannel:0x1';
END_IF
IF (nState_TsGroup1 = 3) THEN 	//Module Error
	
END_IF

IF bSafety_FBErr THEN	//Function block Error
	//Check each FB state
		fbTsFBEdmState(nState:=nState_TsFBEDM);
		sState_TsFBEDM := fbTsFBEdmState.sState;
		IF (nState_TsFBEDM = 4) THEN		//if the safeEDM is in state Error then the Diag-Bits get checked
			fbTsFBEdmDiag(nDiag:=nDiag_TsFBEDM);
			sDiag_TsFBEDM := fbTsFBEdmDiag.sDiag;
		END_IF
		
		fbTsFBEstopState(nState:=nState_TsFBEstop);
		sState_TsFBEstop := fbTsFBEstopState.sState;
		IF (nState_TsFBEstop = 4) THEN		//if the safeEStop is in state Error then the Diag-Bits get checked
			fbTsFBEstopDiag(nDiag:=nDiag_TsFBEstop);
			sDiag_TsFBEstop := fbTsFBEstopDiag.sDiag;
		END_IF
		
		fbTsFBMonState(nState:=nState_TsFBMon);
		sState_TsFBMon := fbTsFBMonState.sState;
		IF (nState_TsFBMon = 4) THEN		//if the safeMon is in state Error then the Diag-Bits get checked
			fbTsFBMonDiag(nDiag:=nDiag_TsFBMon);
			sDiag_TsFBMon := fbTsFBMonDiag.sDiag;
		END_IF
END_IF

IF bSafety_ComErr THEN	//Communication Error
	//Check each TwinSAFE connection state
		//EL1904
		fbTsConnectionState(nState:=nState_EL1904);
		sState_EL1904 := fbTsConnectionState.sState;
		fbTsConnectionDiag(nDiag:=nDiag_EL1904);
		sDiagPart1_EL1904 := fbTsConnectionDiag.sDiagPart1;
		sDiagPart2_EL1904 := fbTsConnectionDiag.sDiagPart2;
		IF (nState_EL1904 = 100) OR (nState_EL1904 = 101) OR (nState_EL1904 = 102) OR (nState_EL1904 = 103) THEN //if the connection is in state RESET, SESSION, CONNECTION or PARAMETER then the EtherCAT state, WcState and CoE-Objects 800E get checked
			IF nEtherCATState_EL1904 = 8 THEN
				IF bWcState_EL1904 THEN
					sErrorText_EL1904 := CONCAT(sErrorText_EL1904, 'The terminal EL1904 has a WcState Error');
				ELSE
					//read CoE-diagnostic-objects 800E
					sMasterNetID := F_CreateAmsNetId(MasterAmsNetID);
					fbEcCoeSdoRead(
							sNetId			:= 	sMasterNetID,	//needs to be changed according to the NetId of the EtherCAT Master
							nSlaveAddr		:= 	1003,				//needs to be changed according to the EtherCAT Addr of the EtherCAT Slave
							nSubIndex		:= 	1,
							nIndex			:= 	16#800E,
							pDstBuf			:= 	ADR(stDiagObjects),
							cbBufLen		:= 	SIZEOF(stDiagObjects),
							bExecute		:= 	TRUE,
							tTimeout		:= 	DEFAULT_ADS_TIMEOUT,
							bCompleteAccess	:= 	TRUE);
					
					IF NOT fbEcCoeSdoRead.bBusy AND NOT fbEcCoeSdoRead.bError THEN
						fbEcCoeSdoRead(bExecute := FALSE);
						fbCoEDiagObjectsEL1904(stDiagObjectsEL1904:=stDiagObjects);	
					ELSIF NOT fbEcCoeSdoRead.bBusy AND fbEcCoeSdoRead.bError THEN
						sErrorText_EL1904 := CONCAT(sErrorText_EL1904, 'Error reading CoE objects of terminal EL1904'); //noch um Platzhalter mit Namen der Klemme ersetzen
					END_IF
					
				END_IF
				
			ELSE
				sErrorText_EL1904 := CONCAT(sErrorText_EL1904, 'The terminal EL1904 is not in the EtherCAT state OP');
			END_IF
			
		END_IF
		
		//EL1918
		// 1. State-Text über FB generieren
	fbTsConnectionStateEL1918(nEtherCATState := nEtherCATState_EL1918);
	sState_EL1918 := fbTsConnectionStateEL1918.sEtherCATState;

		// 2. Diagnose-Text(e) über FB generieren
	fbTsConnectionDiagEL1918(nDiagCode := nEtherCATState_EL1918);
	sDiagPart2_EL1918 := fbTsConnectionDiagEL1918.sDiag;
		
		IF (nState_EL1918 = 100) OR (nState_EL1918 = 101) OR (nState_EL1918 = 102) OR (nState_EL1918 = 103) THEN //if the connection is in state RESET, SESSION, CONNECTION or PARAMETER then the EtherCAT state, WcState and CoE-Objects 800E get checked
			IF nEtherCATState_EL1918 = 8 THEN
				IF bWcState_EL1918 THEN
					sErrorText_EL1918 := CONCAT(sErrorText_EL1918, 'The terminal EL1918 has a WcState Error');
				ELSE
					//read CoE-diagnostic-objects 800E
					sMasterNetID := F_CreateAmsNetId(MasterAmsNetID);
					fbEcCoeSdoRead(
							sNetId			:= 	sMasterNetID,	//needs to be changed according to the NetId of the EtherCAT Master
							nSlaveAddr		:= 	1003,				//needs to be changed according to the EtherCAT Addr of the EtherCAT Slave
							nSubIndex		:= 	1,
							nIndex			:= 	16#800E,
							pDstBuf			:= 	ADR(stDiagObjectsEL1918),
							cbBufLen		:= 	SIZEOF(stDiagObjectsEL1918),
							bExecute		:= 	TRUE,
							tTimeout		:= 	DEFAULT_ADS_TIMEOUT,
							bCompleteAccess	:= 	TRUE);
					
					IF NOT fbEcCoeSdoRead.bBusy AND NOT fbEcCoeSdoRead.bError THEN
						fbEcCoeSdoRead(bExecute := FALSE);
						fbCoEDiagObjectsEL1918(stDiagObjectsEL1918:=stDiagObjectsEL1918);	
					ELSIF NOT fbEcCoeSdoRead.bBusy AND fbEcCoeSdoRead.bError THEN
						sErrorText_EL1918 := CONCAT(sErrorText_EL1918, 'Error reading CoE objects of terminal EL1918'); //noch um Platzhalter mit Namen der Klemme ersetzen
					END_IF
					
				END_IF
				
			ELSE
				sErrorText_EL1918 := CONCAT(sErrorText_EL1918, 'The terminal EL1918 is not in the EtherCAT state OP');
			END_IF
			
		END_IF
		
		//EL2904
		fbTsConnectionState(nState:=nState_EL2904);
		sState_EL2904 := fbTsConnectionState.sState;
		fbTsConnectionDiag(nDiag:=nDiag_EL2904);
		sDiagPart1_EL2904 := fbTsConnectionDiag.sDiagPart1;
		sDiagPart2_EL2904 := fbTsConnectionDiag.sDiagPart2;
		IF (nState_EL2904 = 100) OR (nState_EL2904 = 101) OR (nState_EL2904 = 102) OR (nState_EL2904 = 103) THEN //if the connection is in state RESET, SESSION, CONNECTION or PARAMETER then the EtherCAT state, WcState and CoE-Objects 800E get checked
			IF nEtherCATState_EL2904 = 8 THEN
				IF bWcState_EL2904 THEN
					sErrorText_EL2904 := CONCAT(sErrorText_EL2904, 'The terminal EL2904 has a WcState Error');
				ELSE
					//read CoE-diagnostic-objects 800E
					sMasterNetID := F_CreateAmsNetId(MasterAmsNetID);
					fbEcCoeSdoRead(
							sNetId			:= 	sMasterNetID,	//needs to be changed according to the NetId of the EtherCAT Master
							nSlaveAddr		:= 	1003,				//needs to be changed according to the EtherCAT Addr of the EtherCAT Slave
							nSubIndex		:= 	1,
							nIndex			:= 	16#800E,
							pDstBuf			:= 	ADR(stDiagObjectsEL2904),
							cbBufLen		:= 	SIZEOF(stDiagObjectsEL2904),
							bExecute		:= 	TRUE,
							tTimeout		:= 	DEFAULT_ADS_TIMEOUT,
							bCompleteAccess	:= 	TRUE);
					
					IF NOT fbEcCoeSdoRead.bBusy AND NOT fbEcCoeSdoRead.bError THEN
						fbEcCoeSdoRead(bExecute := FALSE);
						fbCoEDiagObjectsEL2904(stDiagObjectsEL2904:=stDiagObjectsEL2904);	
					ELSIF NOT fbEcCoeSdoRead.bBusy AND fbEcCoeSdoRead.bError THEN
						sErrorText_EL2904 := CONCAT(sErrorText_EL2904, 'Error reading CoE objects of terminal EL2904'); //noch um Platzhalter mit Namen der Klemme ersetzen
					END_IF
					
				END_IF
				
			ELSE
				sErrorText_EL2904 := CONCAT(sErrorText_EL2904, 'The terminal EL2904 is not in the EtherCAT state OP');
			END_IF
			
		END_IF
		
		//EL2912
			// 1. State-Text über FB generieren
	fbTsConnectionStateEL2912(nEtherCATState := nState_EL2912);
	sState_EL1918 := fbTsConnectionStateEL1918.sEtherCATState;

		// 2. Diagnose-Text(e) über FB generieren
	fbTsConnectionDiagEL2912(nDiagCode := nDiag_EL2912);
	sDiagTextEL2912 := fbTsConnectionDiagEL2912.sDiag;
	
		fbTsConnectionState(nState:=nState_EL2912);
		sState_EL2912 := fbTsConnectionState.sState;
		fbTsConnectionDiag(nDiag:=nDiag_EL2904);
		sDiagPart1_EL2912 := fbTsConnectionDiag.sDiagPart1;
		sDiagPart2_EL2912 := fbTsConnectionDiag.sDiagPart2;
		IF (nState_EL2912 = 100) OR (nState_EL2912 = 101) OR (nState_EL2912 = 102) OR (nState_EL2912 = 103) THEN //if the connection is in state RESET, SESSION, CONNECTION or PARAMETER then the EtherCAT state, WcState and CoE-Objects 800E get checked
			IF nEtherCATState_EL2912 = 8 THEN
				IF bWcState_EL2912_1 OR bWcState_EL2912_2 THEN
					sErrorText_EL2912 := CONCAT(sErrorText_EL2912, 'The terminal EL2912 has a WcState Error');
				ELSE
					// 1. State-Text über FB generieren
						fbTsConnectionStateEL2912(nEtherCATState := nState_EL2912);
						sState_EL1918 := fbTsConnectionStateEL1918.sEtherCATState;

					// 2. Diagnose-Text(e) über FB generieren
						fbTsConnectionDiagEL2912(nDiagCode := nDiag_EL2912);
						sDiagTextEL2912 := fbTsConnectionDiagEL2912.sDiag;
					
				END_IF
				
			ELSE
				sErrorText_EL2912 := CONCAT(sErrorText_EL2912, 'The terminal EL2912 is not in the EtherCAT state OP');
			END_IF
			
		END_IF
		//continue with the rest of the terminals...
		
END_IF

	
































//////////////////////////////////////////////////////Analog/////////////////////////////////////////////////////////////////////////////////

//Dogan


 // Zeit immer aktualisieren
tNow := TIME();

// Rising edge von bExecute → Initialisierung
IF (bExecute AND NOT bLastExecute) THEN
    fTime := 0.0;
    tLastCycle := tNow;
    bOut := FALSE;
END_IF
bLastExecute := bExecute;

// Wenn bExecute nicht aktiv → Ausgang 0
IF NOT bExecute THEN
    nOutV1 := 0;
    RETURN;
END_IF

// Zykluszeit berechnen
IF tLastCycle <> T#0S THEN
    fTime := fTime + TO_REAL(TIME_TO_DINT(tNow - tLastCycle)) / 1000.0;
END_IF;
tLastCycle := tNow;

// Signal wählen
CASE SignalMode OF

    SignalMode_Off:
        nOutV1 := 0;

    SignalMode_Static:
        nOutV1 := 3280;
		nOutA1 := 10000;

    SignalMode_Rectangle:
        tOn(IN := TRUE, PT := T#1500MS);
        IF tOn.Q THEN
            bOut := NOT bOut;
            tOn(IN := FALSE);
        ELSE
            tOn(IN := TRUE);
        END_IF;

        IF bOut THEN
            nOutV1 := 30000;
			nOutA1 := 20000;
        ELSE
            nOutV1 := 0;
			nOutA1 := 0;
        END_IF;

    SignalMode_Sinus:
        fSinusValue := fAmplitude * SIN(2.0 * 3.1415926535 * fFrequency * fTime) + fOffset;
        nOutV1 := REAL_TO_INT(fSinusValue);
		nOutA1 := REAL_TO_INT(fSinusValue)/2;
		
SignalMode_Triangle:
	
// Steigung berechnen
fSlope := (4.0 * fAmplitude) / fPeriod;

// Phase berechnen (Ersatz für MOD)
fPhase := fTime - fPeriod * DINT_TO_REAL(TRUNC(fTime / fPeriod));


// Dreiecksignal berechnen
fTriangle := fSlope * ABS(fPhase - (fPeriod / 2.0)) - fAmplitude;

// Ausgang setzen
nOutV1 := REAL_TO_INT(fTriangle + fOffset);
	
    ELSE
        nOutV1 := 0;

END_CASE;

// Fehlerbits

IF bExecute THEN
    AI3174_Error := EL3174.MDP5001_300_Input.MDP5001_300_AI_Standard_Channel_1_Status.Error;

    IF EL3174.MDP5001_300_Input.MDP5001_300_AI_Standard_Channel_1_Status.Overrange THEN
        AI3174_Overrange := TRUE;
    ELSE
        AI3174_Overrange := FALSE;
    END_IF

    IF EL3174.MDP5001_300_Input.MDP5001_300_AI_Standard_Channel_1_Status.Underrange THEN
        AI3174_Underrange := TRUE;
    ELSE
        AI3174_Underrange := FALSE;
    END_IF
ELSE
    AI3174_Error      := FALSE;
    AI3174_Overrange  := FALSE;
    AI3174_Underrange := FALSE;
END_IF

IF bExecute THEN
    EL3074_Error := el3074.MDP5001_300_Input.MDP5001_300_AI_Standard_Channel_1_Status.Error;

    IF EL3074.MDP5001_300_Input.MDP5001_300_AI_Standard_Channel_1_Status.Overrange THEN
        EL3074_Overrange := TRUE;
    ELSE
        EL3074_Overrange := FALSE;
    END_IF

    IF EL3074.MDP5001_300_Input.MDP5001_300_AI_Standard_Channel_1_Status.Underrange THEN
        EL3074_Underrange := TRUE;
    ELSE
        EL3074_Underrange := FALSE;
    END_IF
ELSE
    EL3074_Error      := FALSE;
    EL3074_Overrange  := FALSE;
    EL3074_Underrange := FALSE;
END_IF

IF bExecute THEN
    EL3202_Error := el3202.MDP5001_320_Input.MDP5001_320_RTD_Inputs_Channel_1_Status.Error;

    IF el3202.MDP5001_320_Input.MDP5001_320_RTD_Inputs_Channel_1_Status.Overrange THEN
        EL3202_Overrange := TRUE;
    ELSE
        EL3202_Overrange := FALSE;
    END_IF

    IF el3202.MDP5001_320_Input.MDP5001_320_RTD_Inputs_Channel_1_Status.Underrange THEN
        EL3202_Underrange := TRUE;
    ELSE
        EL3202_Underrange := FALSE;
    END_IF
ELSE
    EL3202_Error      := FALSE;
    EL3202_Overrange  := FALSE;
    EL3202_Underrange := FALSE;
END_IF

IF bExecute THEN
    EL3074_Error := el3074.MDP5001_300_Input.MDP5001_300_AI_Standard_Channel_1_Status.Error;

    IF EL3074.MDP5001_300_Input.MDP5001_300_AI_Standard_Channel_1_Status.Overrange THEN
        EL3074_Overrange := TRUE;
    ELSE
        EL3074_Overrange := FALSE;
    END_IF

    IF EL3074.MDP5001_300_Input.MDP5001_300_AI_Standard_Channel_1_Status.Underrange THEN
        EL3074_Underrange := TRUE;
    ELSE
        EL3074_Underrange := FALSE;
    END_IF
ELSE
    EL3074_Error      := FALSE;
    EL3074_Overrange  := FALSE;
    EL3074_Underrange := FALSE;
END_IF

IF bExecute THEN
    ELM3142_Error := elm3142.MDP5001_350_Input.MDP5001_350_PAI_Status_Channel_1_Status.Error;

    IF ELM3142.MDP5001_350_Input.MDP5001_350_PAI_Status_Channel_1_Status.Overrange THEN
        ELM3142_Overrange := TRUE;
    ELSE
        ELM3142_Overrange := FALSE;
    END_IF

    IF elm3142.MDP5001_350_Input.MDP5001_350_PAI_Status_Channel_1_Status.Underrange THEN
        ELM3142_Underrange := TRUE;
    ELSE
        ELM3142_Underrange := FALSE;
    END_IF
ELSE
    ELM3142_Error      := FALSE;
    ELM3142_Overrange  := FALSE;
    ELM3142_Underrange := FALSE;
END_IF

// Umrechnung in Ampere
IF nIn3174A1 < 0 THEN 
	nCurr:=0;
ELSE
	nCurr:=  nIn3174A1 * 16.0 / 30518 +4; //Extended Range 
END_IF
IF nELM > 0 THEN
		nElmCurr:= nELM * 16.0/7812500+4; // Strom im Messbereich 4..20 mA
ELSE
			nElmCurr := 0;
END_IF
// Umrechnung RTD

	nRTDVal:=  nRTD / 10.0;

// Umrechnung in Volt

	nVoltELM := nELM / 7812500.0 * 10;  // Extended Range
	nVoltEL := 10.0 * nIn3074V1 / 32767;
		
	
//	Alarm

IF bClearLoggedEvents THEN
   bClearLoggedEvents:= NOT fbEventlogger.ClearLoggedEvents(0);
END_IF

(*
IF NOT bIsInitalized THEN
	bIsInitalized := TRUE;
	fbMessage.CreateEx(TC_Events.MyEvents.Start, 0);
	fbAlarm.CreateEx(TC_Events.MyEvents.Stop, TRUE, 0);
END_IF

IF bMessage THEN
	bMessage := FALSE;
	fbMessage.Send(0);
END_IF

IF bAlarm THEN
	bAlarm := FALSE;
	fbAlarm.Raise(0);
END_IF

IF bClearAlarm THEN
	bClearAlarm := FALSE;
	fbAlarm.Clear(0, TRUE);
END_IF
*)

*)



































































//////////////////////////////////////////////////////Motion/////////////////////////////////////////////////////////////////////////////////

//Kuba

//Achsstruktur zyklisch lesen
Axis1.ReadStatus();
//AXIS1 STARTEN

fbPower(
	Axis:= Axis1, 
	Enable:= bEnable, 
	Enable_Positive:= bEnable, 
	Enable_Negative:= bEnable, 
	Override:= , 
	BufferMode:= , 
	Options:= , 
	Status=> , 
	Busy=> , 
	Error=> , 
	ErrorID=> );

fbMoveVelocity(
	Axis:= Axis1, 
	Execute:= bMove, 
	Velocity:= nVelocity, 
	Acceleration:= nDynamik, 
	Deceleration:= nDynamik, 
	Jerk:= , 
	Direction:= , 
	BufferMode:= , 
	Options:= , 
	InVelocity=> , 
	Busy=> , 
	Active=> , 
	CommandAborted=> , 
	Error=> , 
	ErrorID=> );
	
fbReset(
	Axis:= Axis1, 
	Execute:= bReset, 
	Done=> , 
	Busy=> , 
	Error=> , 
	ErrorID=> );
	
//AXIS1 FEHLERMELDUNG	

fbReadDiag( 
	bEnable:= bRead, 
	bAck:= , 
	tTimeout:= , 
	tReadInterval:= , 
	stOptions:= , 
	aDiagHistory:= aMessages, 
	bBusy=> , 
	bValid=> , 
	bError=> , 
	hrErrorCode=> , 
	ipErrorMessage=> , 
	stInfo=> , 
	refAxis:= Axis1);
	
	
//AXIS2 STARTEN
Axis2.ReadStatus();

fbPower2(
	Axis:= Axis2, 
	Enable:= bEnable2, 
	Enable_Positive:= bEnable2, 
	Enable_Negative:= bEnable2, 
	Override:= , 
	BufferMode:= , 
	Options:= , 
	Status=> , 
	Busy=> , 
	Error=> , 
	ErrorID=> );
	
fbMoveVelocity2(
	Axis:= Axis2, 
	Execute:= bMove2, 
	Velocity:= nVelocity, 
	Acceleration:= nDynamik2, 
	Deceleration:= nDynamik2, 
	Jerk:= , 
	Direction:= , 
	BufferMode:= , 
	Options:= , 
	InVelocity=> , 
	Busy=> , 
	Active=> , 
	CommandAborted=> , 
	Error=> , 
	ErrorID=> );
	
fbReset2(
	Axis:= Axis2, 
	Execute:= bReset2, 
	Done=> , 
	Busy=> , 
	Error=> , 
	ErrorID=> );
	
//AXIS2 FEHLERMELDUNG

fbReadDiag2( 
	bEnable:= bRead2, 
	bAck:= , 
	tTimeout:= , 
	tReadInterval:= , 
	stOptions:= , 
	aDiagHistory:= aMessages2, 
	bBusy=> , 
	bValid=> , 
	bError=> , 
	hrErrorCode=> , 
	ipErrorMessage=> , 
	stInfo=> , 
	refAxis:= Axis2);
	
	
	
	
CASE nCase OF 
	0: //INIT
	bMove := FALSE;
	bEnable := FALSE;
	bReset := FALSE;
	IF bStartSequence THEN
		bStartSequence := FALSE;
		nCase := nCase +10;
	END_IF
	
	10: //enable axis
	bEnable := TRUE;
	IF Axis1.Status.ControlLoopClosed THEN
		nCase := nCase +10;
	END_IF
	
	20: //Move
	bMove := TRUE;
	
	99: //
	bMove := FALSE;
	bReset := TRUE;
	IF NOT axis1.Status.Error THEN
		nCase := 0;
	END_IF
END_CASE
IF Axis1.Status.Error OR fbMoveVelocity.Error THEN
	ncase := 99; //error case
END_IF


CASE nCase2 OF 
	0: //INIT
	bMove2 := FALSE;
	bEnable2 := FALSE;
	bReset2 := FALSE;
	IF bStartSequence2 THEN
		bStartSequence2 := FALSE;
		nCase2 := nCase2 +10;
	END_IF
	
	10: //enable axis
	bEnable2 := TRUE;
	IF Axis2.Status.ControlLoopClosed THEN
		nCase2 := nCase2 +10;
	END_IF
	
	20: //Move
	bMove2 := TRUE;
	
	99: //
	bMove2 := FALSE;
	bReset2 := TRUE;
	IF NOT Axis2.Status.Error THEN
		nCase2 := 0;
	END_IF
END_CASE
IF Axis2.Status.Error OR fbMoveVelocity2.Error THEN
	ncase2 := 99; //error case
END_IF

END_PROGRAM

// ---- POUs/TwinSAFE FBs/FB_CoEDiagObjects_EL1904.TcPOU
FUNCTION_BLOCK FB_CoEDiagObjects_EL1904
VAR_INPUT
	stDiagObjectsEL1904 											: ST_TsDiagObjectsEL1904;
END_VAR
VAR_OUTPUT
	sDiagText      : STRING(255);                 // Gesamtausgabe als Sammelstring
	asDiagList     : ARRAY[1..10] OF STRING(120); // Einzelmeldungen
	nDiagCount     : INT;                         // Anzahl aktiver Meldungen
	
END_VAR
VAR
	TsDiagObjectsBitsEL1904_bSensorTestError_Input1			: BOOL;
	TsDiagObjectsBitsEL1904_bSensorTestError_Input2			: BOOL;
	TsDiagObjectsBitsEL1904_bSensorTestError_Input3			: BOOL;
	TsDiagObjectsBitsEL1904_bSensorTestError_Input4			: BOOL;
	TsDiagObjectsBitsEL1904_bErrFirstInputPair 				: BOOL;
	TsDiagObjectsBitsEL1904_bErrSecondInputPair 			: BOOL;
	TsDiagObjectsBitsEL1904_bMatOpModeErrFirstInputPair 	: BOOL;
	TsDiagObjectsBitsEL1904_bMatOpModeErrSecondInputPair 	: BOOL;
	TsDiagObjectsBitsEL1904_bMatOpModeExtSupplyError_Input1 : BOOL;
	TsDiagObjectsBitsEL1904_bMatOpModeExtSupplyError_Input2 : BOOL;
	TsDiagObjectsBitsEL1904_bMatOpModeExtSupplyError_Input3 : BOOL;
	TsDiagObjectsBitsEL1904_bMatOpModeExtSupplyError_Input4 : BOOL;
	i 														: INT;
END_VAR

//Sensor-Test Error
TsDiagObjectsBitsEL1904_bSensorTestError_Input1		:= stDiagObjectsEL1904.nSensorTestError.0;
TsDiagObjectsBitsEL1904_bSensorTestError_Input2		:= stDiagObjectsEL1904.nSensorTestError.1;
TsDiagObjectsBitsEL1904_bSensorTestError_Input3		:= stDiagObjectsEL1904.nSensorTestError.2;
TsDiagObjectsBitsEL1904_bSensorTestError_Input4		:= stDiagObjectsEL1904.nSensorTestError.3;

//Error during two channel evaluation
TsDiagObjectsBitsEL1904_bErrFirstInputPair 			 := stDiagObjectsEL1904.nDuringTwoChannelEvaluationError.0;
TsDiagObjectsBitsEL1904_bErrSecondInputPair 		 := stDiagObjectsEL1904.nDuringTwoChannelEvaluationError.1;

//Error in the safety mat operating mode: input pair disagree
TsDiagObjectsBitsEL1904_bMatOpModeErrFirstInputPair	 := stDiagObjectsEL1904.nMatModeInputPairDisagreeError.0 
																			AND stDiagObjectsEL1904.nMatModeInputPairDisagreeError.1;
TsDiagObjectsBitsEL1904_bMatOpModeErrSecondInputPair := stDiagObjectsEL1904.nMatModeInputPairDisagreeError.2 
																			AND stDiagObjectsEL1904.nMatModeInputPairDisagreeError.3;
																			
//Error in the safety mat operating mode: external supply
TsDiagObjectsBitsEL1904_bMatOpModeExtSupplyError_Input1 := stDiagObjectsEL1904.nMatModeExternalSupplyError.0;
TsDiagObjectsBitsEL1904_bMatOpModeExtSupplyError_Input2 := stDiagObjectsEL1904.nMatModeExternalSupplyError.1;
TsDiagObjectsBitsEL1904_bMatOpModeExtSupplyError_Input3 := stDiagObjectsEL1904.nMatModeExternalSupplyError.2;
TsDiagObjectsBitsEL1904_bMatOpModeExtSupplyError_Input4 := stDiagObjectsEL1904.nMatModeExternalSupplyError.3;


//muss noch um die Ausgabe in Textform über Strings ergänzt werden!
sDiagText := '';
nDiagCount := 0;

FOR i := 1 TO 20 DO
	asDiagList[i] := '';
END_FOR;

IF TsDiagObjectsBitsEL1904_bSensorTestError_Input1 THEN
	nDiagCount := nDiagCount + 1;
	asDiagList[nDiagCount] := 'Sensor Test Error Input1';
	sDiagText := CONCAT(sDiagText, CONCAT(asDiagList[nDiagCount], '; '));
END_IF

IF TsDiagObjectsBitsEL1904_bSensorTestError_Input2 THEN
    nDiagCount := nDiagCount + 1;
    asDiagList[nDiagCount] := 'Sensor Test Error Input2';
    sDiagText := CONCAT(sDiagText, CONCAT(asDiagList[nDiagCount], '; '));
END_IF

IF TsDiagObjectsBitsEL1904_bSensorTestError_Input3 THEN
    nDiagCount := nDiagCount + 1;
    asDiagList[nDiagCount] := 'Sensor Test Error Input3';
    sDiagText := CONCAT(sDiagText, CONCAT(asDiagList[nDiagCount], '; '));
END_IF

IF TsDiagObjectsBitsEL1904_bSensorTestError_Input4 THEN
    nDiagCount := nDiagCount + 1;
    asDiagList[nDiagCount] := 'Sensor Test Error Input4';
    sDiagText := CONCAT(sDiagText, CONCAT(asDiagList[nDiagCount], '; '));
END_IF

IF TsDiagObjectsBitsEL1904_bErrFirstInputPair THEN
    nDiagCount := nDiagCount + 1;
    asDiagList[nDiagCount] := 'Two-channel evaluation error on first input pair';
    sDiagText := CONCAT(sDiagText, CONCAT(asDiagList[nDiagCount], '; '));
END_IF

IF TsDiagObjectsBitsEL1904_bErrSecondInputPair THEN
    nDiagCount := nDiagCount + 1;
    asDiagList[nDiagCount] := 'Two-channel evaluation error on second input pair';
    sDiagText := CONCAT(sDiagText, CONCAT(asDiagList[nDiagCount], '; '));
END_IF

IF TsDiagObjectsBitsEL1904_bMatOpModeErrFirstInputPair THEN
    nDiagCount := nDiagCount + 1;
    asDiagList[nDiagCount] := 'Safety mat mode: Input pair 1 disagree';
    sDiagText := CONCAT(sDiagText, CONCAT(asDiagList[nDiagCount], '; '));
END_IF

IF TsDiagObjectsBitsEL1904_bMatOpModeErrSecondInputPair THEN
    nDiagCount := nDiagCount + 1;
    asDiagList[nDiagCount] := 'Safety mat mode: Input pair 2 disagree';
    sDiagText := CONCAT(sDiagText, CONCAT(asDiagList[nDiagCount], '; '));
END_IF

IF TsDiagObjectsBitsEL1904_bMatOpModeExtSupplyError_Input1 THEN
    nDiagCount := nDiagCount + 1;
    asDiagList[nDiagCount] := 'Safety mat external supply error Input1';
    sDiagText := CONCAT(sDiagText, CONCAT(asDiagList[nDiagCount], '; '));
END_IF

IF TsDiagObjectsBitsEL1904_bMatOpModeExtSupplyError_Input2 THEN
    nDiagCount := nDiagCount + 1;
    asDiagList[nDiagCount] := 'Safety mat external supply error Input2';
    sDiagText := CONCAT(sDiagText, CONCAT(asDiagList[nDiagCount], '; '));
END_IF

IF TsDiagObjectsBitsEL1904_bMatOpModeExtSupplyError_Input3 THEN
    nDiagCount := nDiagCount + 1;
    asDiagList[nDiagCount] := 'Safety mat external supply error Input3';
    sDiagText := CONCAT(sDiagText, CONCAT(asDiagList[nDiagCount], '; '));
END_IF

IF TsDiagObjectsBitsEL1904_bMatOpModeExtSupplyError_Input4 THEN
    nDiagCount := nDiagCount + 1;
    asDiagList[nDiagCount] := 'Safety mat external supply error Input4';
    sDiagText := CONCAT(sDiagText, CONCAT(asDiagList[nDiagCount], '; '));
END_IF

END_FUNCTION_BLOCK

// ---- POUs/TwinSAFE FBs/FB_TsFBEDM_State.TcPOU
FUNCTION_BLOCK FB_TsFBEDM_State
VAR_INPUT
	nState: USINT;
END_VAR
VAR_OUTPUT
	sState: STRING;
END_VAR
VAR
END_VAR

CASE nState OF
	2:		sState := 'STOP';	
	4:		sState := 'ERROR';	
	5:		sState := 'RESET';	
	14:		sState := 'MON_OFF';	
	15:		sState := 'MON_ON';	
ELSE 
	sState := 'undefined';
END_CASE

END_FUNCTION_BLOCK

// ---- POUs/TwinSAFE FBs/FB_TsFBEDM_Diag.TcPOU
FUNCTION_BLOCK FB_TsFBEDM_Diag
VAR_INPUT
	nDiag		: USINT;
END_VAR
VAR_OUTPUT
	sDiag		: STRING;
END_VAR
VAR
END_VAR

CASE nDiag OF
	0:		sDiag := 'No Error';		
	1:		sDiag := 'Switch-OFF timer elapsed';	
	2:		sDiag := 'Switch-ON timer elapsed';	
ELSE 
	sDiag := 'undefined';
END_CASE

END_FUNCTION_BLOCK

// ---- POUs/TwinSAFE FBs/FB_TsFBEStop_Diag.TcPOU
FUNCTION_BLOCK FB_TsFBEStop_Diag
VAR_INPUT
	nDiag		: UINT;
END_VAR
VAR_OUTPUT
	sDiag		: STRING;
END_VAR
VAR
END_VAR

CASE TO_WORD(nDiag) AND 16#00FF OF
	1:		sDiag := 'Discrepancy error input group 1';		//Bit 0
	2:		sDiag := 'Discrepancy error input group 2';		//Bit 1
	4:		sDiag := 'Discrepancy error input group 3';		//Bit 2
	8:		sDiag := 'Discrepancy error input group 4';		//Bit 3
	16:		sDiag := 'EDM monitoring error EDM1';			//Bit 4
	32:		sDiag := 'EDM monitoring error EDM2';			//Bit 5
END_CASE

CASE TO_WORD(nDiag) AND 16#FF00 OF
	256:	sDiag := CONCAT(sDiag, ' - with activated option "SAFE Inputs after Disc Error"');	//Bit 8
	512:	sDiag := CONCAT(sDiag, ' - with activated option "SAFE Inputs after Disc Error"');	//Bit 9
	1024:	sDiag := CONCAT(sDiag, ' - with activated option "SAFE Inputs after Disc Error"');	//Bit 10
	2048:	sDiag := CONCAT(sDiag, ' - with activated option "SAFE Inputs after Disc Error"');	//Bit 11
END_CASE
	
IF nDiag = 0
THEN
	sDiag := 'No error';
ELSIF sDiag = ''
THEN
	sDiag := 'undefined';		
END_IF

END_FUNCTION_BLOCK

// ---- POUs/TwinSAFE FBs/FB_TsFBMon_State.TcPOU
FUNCTION_BLOCK FB_TsFBMon_State
VAR_INPUT
	nState		: USINT;
END_VAR
VAR_OUTPUT
	sState		: STRING;
END_VAR
VAR
END_VAR

CASE nState OF
	1:		sState := 'RUN';	
	2:		sState := 'STOP';	
	3:		sState := 'SAFE';	
	4:		sState := 'ERROR';	
	5:		sState := 'RESET';	
	6:		sState := 'START';	
	7:		sState := 'ERRORDELAY';	
	8:		sState := 'DELAYOUT';	
	9:		sState := 'FUNCTEST';	
ELSE 
	sState := 'undefined';
END_CASE

END_FUNCTION_BLOCK

// ---- POUs/TwinSAFE FBs/FB_TsConnection_EtherCatState_EL1918.TcPOU
FUNCTION_BLOCK FB_TsConnection_EtherCatState_EL1918
VAR_INPUT
    nEtherCATState : UINT; // EtherCAT Slave State
END_VAR
VAR_OUTPUT
    sEtherCATState : STRING;
END_VAR

CASE nEtherCATState OF
    16#0001: sEtherCATState := 'INIT';
    16#0002: sEtherCATState := 'PREOP';
    16#0003: sEtherCATState := 'BOOT';
    16#0004: sEtherCATState := 'SAFEOP';
    16#0008: sEtherCATState := 'OP';
ELSE
    sEtherCATState := 'undefined';
END_CASE

END_FUNCTION_BLOCK

// ---- POUs/TwinSAFE FBs/FB_TsConnection_Diag_EL1918.TcPOU
FUNCTION_BLOCK FB_TsConnection_Diag_EL1918
VAR_INPUT
    nDiagCode : UINT; // Diagnosecode (Bitfeld)
END_VAR
VAR_OUTPUT
    sDiag : STRING(255);
END_VAR

sDiag := '';

IF (nDiagCode AND 16#0001) <> 0 THEN
    sDiag := CONCAT(sDiag, 'Slave signals error; ');
END_IF;
IF (nDiagCode AND 16#0002) <> 0 THEN
    sDiag := CONCAT(sDiag, 'Invalid vendorId/productCode; ');
END_IF;
IF (nDiagCode AND 16#0004) <> 0 THEN
    sDiag := CONCAT(sDiag, 'Initialization error; ');
END_IF;
IF (nDiagCode AND 16#0008) <> 0 THEN
    sDiag := CONCAT(sDiag, 'Slave disabled; ');
END_IF;
IF (nDiagCode AND 16#0010) <> 0 THEN
    sDiag := CONCAT(sDiag, 'Slave not present; ');
END_IF;
IF (nDiagCode AND 16#0020) <> 0 THEN
    sDiag := CONCAT(sDiag, 'Link error; ');
END_IF;
IF (nDiagCode AND 16#0040) <> 0 THEN
    sDiag := CONCAT(sDiag, 'Missing link; ');
END_IF;
IF (nDiagCode AND 16#0080) <> 0 THEN
    sDiag := CONCAT(sDiag, 'Unexpected link; ');
END_IF;
IF (nDiagCode AND 16#0100) <> 0 THEN
    sDiag := CONCAT(sDiag, 'Comm Port A; ');
END_IF;
IF (nDiagCode AND 16#0200) <> 0 THEN
    sDiag := CONCAT(sDiag, 'Comm Port B; ');
END_IF;
IF (nDiagCode AND 16#0400) <> 0 THEN
    sDiag := CONCAT(sDiag, 'Comm Port C; ');
END_IF;
IF (nDiagCode AND 16#0800) <> 0 THEN
    sDiag := CONCAT(sDiag, 'Comm Port D; ');
END_IF;

END_FUNCTION_BLOCK

// ---- POUs/TwinSAFE FBs/FB_TsConnection_EtherCATState_EL2904.TcPOU
FUNCTION_BLOCK FB_TsConnection_EtherCATState_EL2904
VAR_INPUT
    nEtherCATState : UINT; // EtherCAT Slave State
END_VAR
VAR_OUTPUT
    sEtherCATState : STRING;
END_VAR

CASE nEtherCATState OF
    16#0001: sEtherCATState := 'INIT';
    16#0002: sEtherCATState := 'PREOP';
    16#0003: sEtherCATState := 'BOOT';
    16#0004: sEtherCATState := 'SAFEOP';
    16#0008: sEtherCATState := 'OP';
ELSE
    sEtherCATState := 'undefined';
END_CASE

END_FUNCTION_BLOCK

// ---- POUs/TwinSAFE FBs/FB_TsConnection_EtherCATState_EL2912.TcPOU
FUNCTION_BLOCK FB_TsConnection_EtherCATState_EL2912
VAR_INPUT
    nEtherCATState : UINT; // EtherCAT Slave State
END_VAR
VAR_OUTPUT
    sEtherCATState : STRING;
END_VAR

CASE nEtherCATState OF
    16#0001: sEtherCATState := 'INIT';
    16#0002: sEtherCATState := 'PREOP';
    16#0003: sEtherCATState := 'BOOT';
    16#0004: sEtherCATState := 'SAFEOP';
    16#0008: sEtherCATState := 'OP';
ELSE
    sEtherCATState := 'undefined';
END_CASE

END_FUNCTION_BLOCK

// ---- POUs/TwinSAFE FBs/FB_TsConnection_Diag_EL2912.TcPOU
FUNCTION_BLOCK FB_TsConnection_Diag_EL2912
VAR_INPUT
    nDiagCode : UINT; // Diagnosecode (Bitfeld)
END_VAR
VAR_OUTPUT
    sDiag : STRING(255);
END_VAR

sDiag := '';

IF (nDiagCode AND 16#0001) <> 0 THEN
    sDiag := CONCAT(sDiag, 'Slave signals error; ');
END_IF;
IF (nDiagCode AND 16#0002) <> 0 THEN
    sDiag := CONCAT(sDiag, 'Invalid vendorId/productCode; ');
END_IF;
IF (nDiagCode AND 16#0004) <> 0 THEN
    sDiag := CONCAT(sDiag, 'Initialization error; ');
END_IF;
IF (nDiagCode AND 16#0008) <> 0 THEN
    sDiag := CONCAT(sDiag, 'Slave disabled; ');
END_IF;
IF (nDiagCode AND 16#0010) <> 0 THEN
    sDiag := CONCAT(sDiag, 'Slave not present; ');
END_IF;
IF (nDiagCode AND 16#0020) <> 0 THEN
    sDiag := CONCAT(sDiag, 'Link error; ');
END_IF;
IF (nDiagCode AND 16#0040) <> 0 THEN
    sDiag := CONCAT(sDiag, 'Missing link; ');
END_IF;
IF (nDiagCode AND 16#0080) <> 0 THEN
    sDiag := CONCAT(sDiag, 'Unexpected link; ');
END_IF;
IF (nDiagCode AND 16#0100) <> 0 THEN
    sDiag := CONCAT(sDiag, 'Comm Port A; ');
END_IF;
IF (nDiagCode AND 16#0200) <> 0 THEN
    sDiag := CONCAT(sDiag, 'Comm Port B; ');
END_IF;
IF (nDiagCode AND 16#0400) <> 0 THEN
    sDiag := CONCAT(sDiag, 'Comm Port C; ');
END_IF;
IF (nDiagCode AND 16#0800) <> 0 THEN
    sDiag := CONCAT(sDiag, 'Comm Port D; ');
END_IF;

END_FUNCTION_BLOCK
